// TIA Portal V20 export
TYPE "typeEmHomedCheck"
// stored: Access Published, Namespace Unit1.Em6
   STRUCT
      cmVisionUnitAxisZ : Bool;
      cmVisionPusherSupportUpDown : Bool;
      cmVisionTriggerSensor : Bool;
      cmVisionController : Bool;
      cmQrReader : Bool;
      cmQrReadHandy : Bool;
   END_STRUCT;
END_TYPE
